ABB RobotStudio station: Attempt.rspag

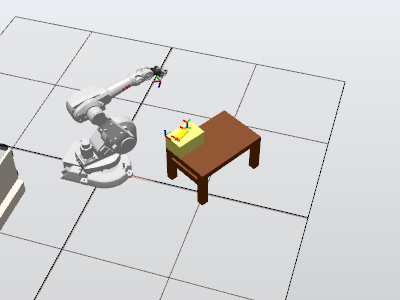
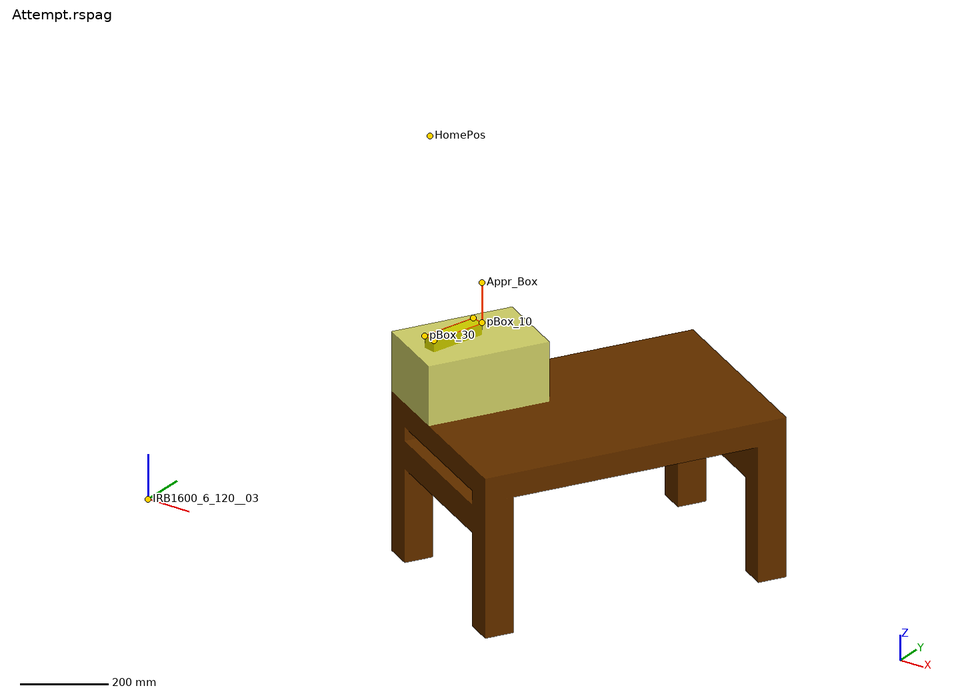
[picture v1: parts stored in the station drawn from their meshes, with robot base, taught points and paths (robot models come from the ABB library and are not in the file)]
--- station ---
Station Station (saved by RobotStudio 25.2.11266.1)
Controller Controller1
  mechanical unit ROB_1: IRB1600_6_120__03, 6 joints, base frame (0, 0, 0) mm
Layout (positions relative to the parent item):
  - IRB1600_6_120__03 [mechanism, from %ABB.RobotStudio.Models.IRB1600%\IRB1600_6_120_G_03.rslib] at (0, 0, 0) mm; joint values [0.8727, -0.5236, 0.3491, 0, 0.5236, 0] (rad or m)
  - Pen [mechanism, from Library\Pen.rslib] at (362.83, 432.41, 979.82) mm, rotated rx -180 ry 70 rz -130 deg
  - IRC5_Control-Module [part, from %ABB.RobotStudio.Models.IRC5%\IRC5_Control-Module.rslib] at (-759.17, -894.97, 100) mm, rotated rx 90 ry 0 rz 90 deg
  - Table [part] at (600, 100, 0) mm, rotated rx 0 ry 0 rz -30 deg, size 500 x 750 x 400 mm
  - Box [part] at (600, 100, 400) mm, rotated rx 0 ry 0 rz -30 deg, size 200 x 300 x 180 mm
Attachment: Pen is attached to IRB1600_6_120__03 / Link6

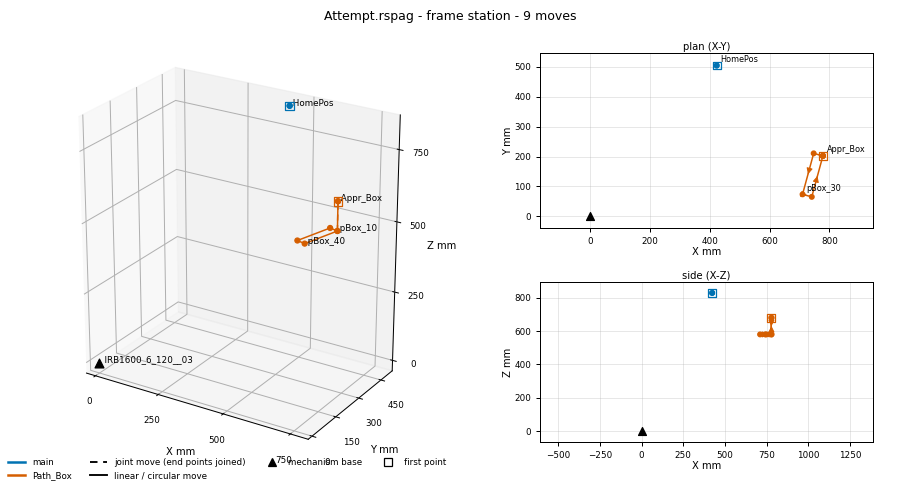
[picture p0: tool path of Attempt.rspag in frame station, 9 of 9 moves have a stored position in this frame; points joined in program order, loops and branches not executed]
--- Backups/Controller1/RAPID/TASK1/PROGMOD/CalibData.mod ---
MODULE CalibData
    PERS tooldata Pen_TCP:=[TRUE,[[110,0,140],[0.707106781,0,0.707106781,0]],[1,[10.7435139,0,140],[1,0,0,0],0,0,0]];
    TASK PERS wobjdata Wobj_Box:=[FALSE,TRUE,"",[[599.999783494,100.000125,550],[0.9659258,0,0,-0.258819143]],[[0,0,0],[1,0,0,0]]];
ENDMODULE

--- Backups/Controller1/RAPID/TASK1/PROGMOD/Module1.mod ---
MODULE Module1
    CONST robtarget Target_10:=[[103.446463924,177.777860178,30],[0,-0.130526293,0.991444848,0],[0,-2,1,0],[9E+09,9E+09,9E+09,9E+09,9E+09,9E+09]];
    CONST robtarget Target_20:=[[72.510503038,169.594512816,30],[0,-0.130526293,0.991444848,0],[0,-2,1,0],[9E+09,9E+09,9E+09,9E+09,9E+09,9E+09]];
    CONST robtarget Target_30:=[[108.824546102,32.316800767,30],[0,-0.130526293,0.991444848,0],[0,-2,1,0],[9E+09,9E+09,9E+09,9E+09,9E+09,9E+09]];
    CONST robtarget Target_40:=[[139.760506988,40.50014813,30],[0,-0.130526293,0.991444848,0],[0,-2,1,0],[9E+09,9E+09,9E+09,9E+09,9E+09,9E+09]];
    CONST robtarget Appr_Box:=[[103.446463924,177.777860178,130],[0,-0.130526293,0.991444848,0],[0,-2,1,0],[9E+09,9E+09,9E+09,9E+09,9E+09,9E+09]];
    CONST robtarget pBox_10:=[[103.446463924,177.777860178,30],[0,-0.130526293,0.991444848,0],[0,-2,1,0],[9E+09,9E+09,9E+09,9E+09,9E+09,9E+09]];
    CONST robtarget pBox_20:=[[72.510503038,169.594512816,30],[0,-0.130526293,0.991444848,0],[0,-2,1,0],[9E+09,9E+09,9E+09,9E+09,9E+09,9E+09]];
    CONST robtarget pBox_30:=[[108.824546102,32.316800767,30],[0,-0.130526293,0.991444848,0],[0,-2,1,0],[9E+09,9E+09,9E+09,9E+09,9E+09,9E+09]];
    CONST robtarget pBox_40:=[[139.760506988,40.50014813,30],[0,-0.130526293,0.991444848,0],[0,-2,1,0],[9E+09,9E+09,9E+09,9E+09,9E+09,9E+09]];
    CONST robtarget HomePos:=[[423.210991524,504.363219574,828.57065573],[0.157378696,0.416197741,-0.892538935,0.073386891],[0,-1,0,0],[9E+09,9E+09,9E+09,9E+09,9E+09,9E+09]];
    !***********************************************************
    !
    ! Module:  Module1
    !
    ! Description:
    !   <Insert description here>
    !
    ! Author: M220173
    !
    ! Version: 1.0
    !
    !***********************************************************


    !***********************************************************
    !
    ! Procedure main
    !
    !   This is the entry point of your program
    !
    !***********************************************************
    PROC main()
        !Add your code here
        MoveJ HomePos,v300,fine,Pen_TCP\WObj:=wobj0;
        Path_Box;
        MoveJ HomePos,v300,fine,Pen_TCP\WObj:=wobj0;
    ENDPROC
    PROC Path_Box()
        MoveJ Appr_Box,v300,fine,Pen_TCP\WObj:=Wobj_Box;
        MoveL pBox_10,v300,fine,Pen_TCP\WObj:=Wobj_Box;
        MoveL pBox_20,v300,fine,Pen_TCP\WObj:=Wobj_Box;
        MoveL pBox_30,v300,fine,Pen_TCP\WObj:=Wobj_Box;
        MoveL pBox_40,v300,fine,Pen_TCP\WObj:=Wobj_Box;
        MoveL pBox_10,v300,fine,Pen_TCP\WObj:=Wobj_Box;
        MoveJ Appr_Box,v300,fine,Pen_TCP\WObj:=Wobj_Box;
    ENDPROC
ENDMODULE
